Staubli VAL3: iPlate3.pgx

public program iPlate3(num& nNum[] (dimensions=1))
begin
  nNum=dioGet(iPlate3)
end
